// This version uses the EL3161 and it's built in IIR filter
PROGRAM AnalogPrescaledSpeedCalculator
VAR_INPUT
	// Analog speed as 0-10v from PC Pin 13
	iAnalogSpeed AT %I*: INT;
END_VAR
VAR_OUTPUT
	// Demanded spindle speed in RPM
	DemandedSpeed : UINT;
END_VAR

DemandedSpeed := TO_UINT(MIN(24000, MAX(0, iAnalogSpeed)));

END_PROGRAM

(* stored: Version 1.1.0.1, ProductVersion 3.1.4022.16
   POU AnalogPrescaledSpeedCalculator: Id {331e867a-d9f4-4f14-8847-df60cde98080}, SpecialFunc None *)
